// TIA Portal V17 export
// export: Created 2025-03-05T08:01:34.6965232Z, ExportSetting WithDefaults, DisplayName Totally Integrated Automation Portal, DisplayVersion V17 Update 8, DisplayName TIA Portal Openness, DisplayVersion V17 Update 8, DisplayName TIA Portal Version Control Interface, DisplayVersion V17, DisplayName SINAMICS Startdrive Advanced, DisplayVersion V17 SP2, DisplayName SINAMICS Startdrive G110M, G120, G120C, G120D, G120P, G115D, DisplayVersion V17 SP2, DisplayName SINAMICS Startdrive G130, G150, S120, S150, SINAMICS MV, S210, DisplayVersion V17 SP2, DisplayName STEP 7 Professional, DisplayVersion V17 Update 8, DisplayName SINUMERIK ONE STEP 7 Toolbox, DisplayVersion V17 Update 12, DisplayName SINUMERIK 840D sl STEP 7 Toolbox, DisplayVersion V17 Update 12, DisplayName STEP 7 Safety, DisplayVersion V17 Update 6, DisplayName WinCC Advanced, DisplayVersion V17 Update 8
FUNCTION "FC16000_OPC_UA_GENERAL" : Void   // FC16000, LAD
{ S7_Optimized_Access := 'TRUE' }
VERSION : 0.1
// stored: AutoNumber false, IsIECCheckEnabled false, SetENOAutomatically false, UDAEnableTagReadback false
BEGIN

REGION Network 1: <<<<<<<<<<<<<<<<<<<<<<< CLIENTS >>>>>>>>>>>>>>>>>>>>>>>>>
   // -DBs CLIENT DATA seran los que ya existen del DB16001 en adelante (DB16001-DB16007).
   // -Los DBs automaticamente generados en la carpeta SYSTEM BLOCKS > PROGRAM RESOURCES los reordenaremos del DB16101 en adelante (DB16101-DB16107) con los nombres: "DB16101_U01_STA3_MEAS_PC_CLIENT".
   // -Los DBs instancias asociados al bloque OPC_UA_Method_Call_C generados en la carpeta SYSTEM BLOCKS > PROGRAM RESOURCES los reordenaremos del DB16201 en adelante (DB16201-DB16207) con los nombres: "DB16201_U01_STA3_MEAS_CALL_METHOD".
END_REGION

REGION Network 2
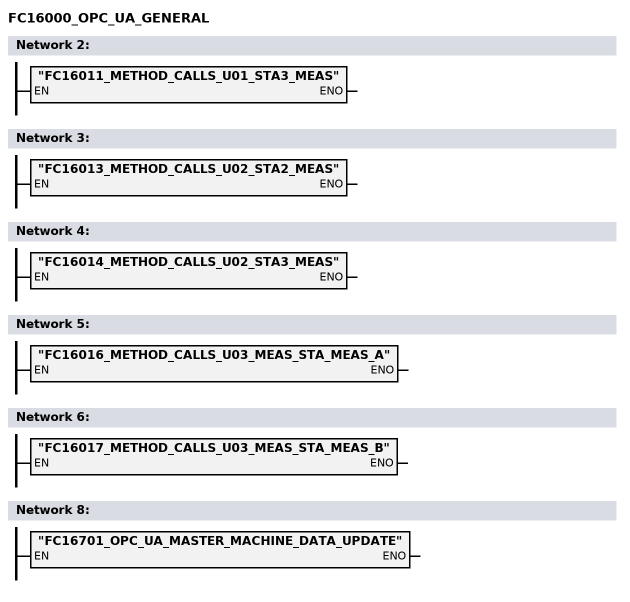
   RUNG wire#powerrail
      "FC16011_METHOD_CALLS_U01_STA3_MEAS"()
   END_RUNG
   // the same network as SCL:
   "FC16011_METHOD_CALLS_U01_STA3_MEAS"();
END_REGION

REGION Network 3
   RUNG wire#powerrail
      "FC16013_METHOD_CALLS_U02_STA2_MEAS"()
   END_RUNG
   // the same network as SCL:
   "FC16013_METHOD_CALLS_U02_STA2_MEAS"();
END_REGION

REGION Network 4
   RUNG wire#powerrail
      "FC16014_METHOD_CALLS_U02_STA3_MEAS"()
   END_RUNG
   // the same network as SCL:
   "FC16014_METHOD_CALLS_U02_STA3_MEAS"();
END_REGION

REGION Network 5
   RUNG wire#powerrail
      "FC16016_METHOD_CALLS_U03_MEAS_STA_MEAS_A"()
   END_RUNG
   // the same network as SCL:
   "FC16016_METHOD_CALLS_U03_MEAS_STA_MEAS_A"();
END_REGION

REGION Network 6
   RUNG wire#powerrail
      "FC16017_METHOD_CALLS_U03_MEAS_STA_MEAS_B"()
   END_RUNG
   // the same network as SCL:
   "FC16017_METHOD_CALLS_U03_MEAS_STA_MEAS_B"();
END_REGION

REGION Network 7: <<<<<<<<<<<<<<<<<<<<<<< MASTER >>>>>>>>>>>>>>>>>>>>>>>>>
END_REGION

REGION Network 8
   RUNG wire#powerrail
      "FC16701_OPC_UA_MASTER_MACHINE_DATA_UPDATE"()
   END_RUNG
   // the same network as SCL:
   "FC16701_OPC_UA_MASTER_MACHINE_DATA_UPDATE"();
END_REGION
END_FUNCTION
